(* IEC 61131-3 sources: Industry-PLC-LLM/data/PLCBEAD_repo/PLCBEAD_PLCEmbed-main/PLC-BEAD/Source/GEB/INT_TO_TIME, 1 file *)

(* ---- INT_TO_TIME.ST ---- *)
FUNCTION _INT_TO_TIME:TIME

	VAR_INPUT
		IN :	INT;
	END_VAR

	_INT_TO_TIME := DINT_TO_TIME(INT_TO_DINT(IN));

END_FUNCTION

PROGRAM program0
	VAR
		IN :	INT;
		OUT : TIME;
	END_VAR

	OUT := _INT_TO_TIME(IN);
END_PROGRAM
